DATA_BLOCK "DB"
{ S7_Optimized_Access := 'false' }
    VAR
        cnt: DINT;
        first: BOOL;
        curTimerValue: TIME;
        state0: STATE;
        curTime: REAL;
        loopsKilled: DINT;
        curTimer: INT;
    END_VAR
BEGIN
    first := TRUE;
END_DATA_BLOCK
